PROGRAM T02_ACCESSORY
VAR
END_VAR

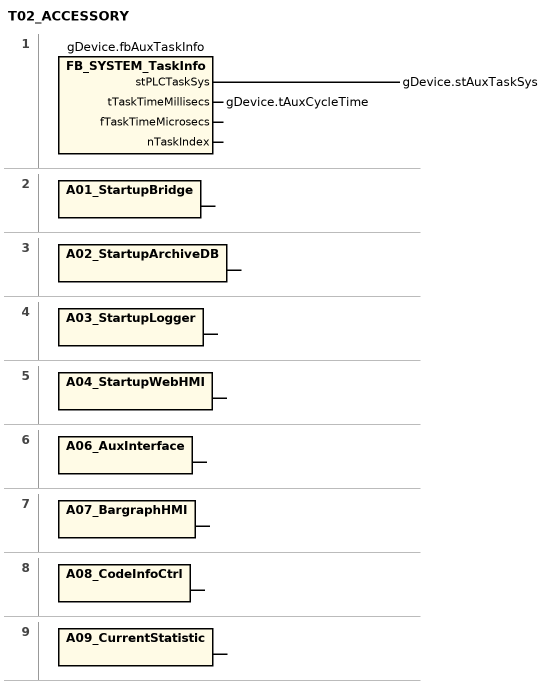
// NETWORK 1
gDevice.fbAuxTaskInfo(tTaskTimeMillisecs => gDevice.tAuxCycleTime); // FB_SYSTEM_TaskInfo
gDevice.stAuxTaskSys := gDevice.fbAuxTaskInfo.stPLCTaskSys;

// NETWORK 2
A01_StartupBridge();

// NETWORK 3
A02_StartupArchiveDB();

// NETWORK 4
A03_StartupLogger();

// NETWORK 5
A04_StartupWebHMI();

// NETWORK 6
A06_AuxInterface();

// NETWORK 7
A07_BargraphHMI();

// NETWORK 8
A08_CodeInfoCtrl();

// NETWORK 9
A09_CurrentStatistic();

END_PROGRAM

(* stored: Version 1.1.0.1
   POU T02_ACCESSORY: Id {6b29b286-a68d-4ab7-9bab-97bad157a82c}, SpecialFunc None *)
